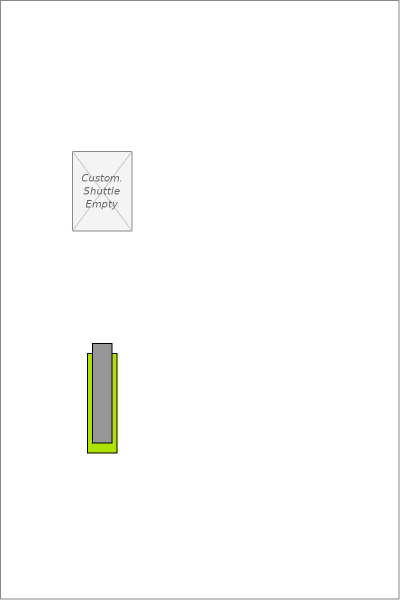
VISUALIZATION VISU_ST170  // 400x600
    Image (72,151 60x80), angle 90, invisible if: NOT __ISVALIDREF(GVL.st170_aut._Mover), image: Custom.Shuttle Empty
    Rectangle (87,353 30x100)
    Rectangle (92,343 20x100)
        p2738717112: -GVL.st170_aut.fb_ABL_RFID.simu_axis170_01Z.rOUT_PixActual
END_VISUALIZATION

// ---- POUs/20_AUTO/ST175/VISU_Recipe_ST175.TcVIS
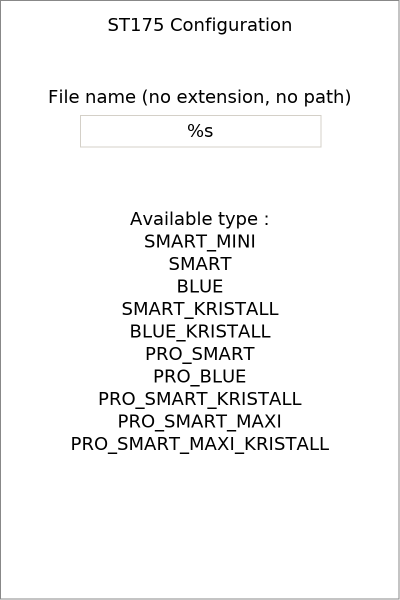
VISUALIZATION VISU_Recipe_ST175  // 400x600
    Textfield (80,115 241x32), "%s", text variable: _20_AUTO.recipe.st175.file_name
        OnMouseDown: write the text variable via Default
    Label (0,5 400x40), "ST175 Configuration"
    Label (24,87 352x20), "File name (no extension, no path)"
    Label (59,177 282x309), "Available type : SMART_MINI SMART BLUE SMART_KRISTALL BLUE_KRISTALL PRO_SMART PRO_BLUE PRO_SMART_KRISTALL PRO_SMART_MAXI PRO_SMART_MAXI_KRISTALL"
END_VISUALIZATION

// ---- POUs/20_AUTO/ST180/VISU_Recipe_ST180.TcVIS
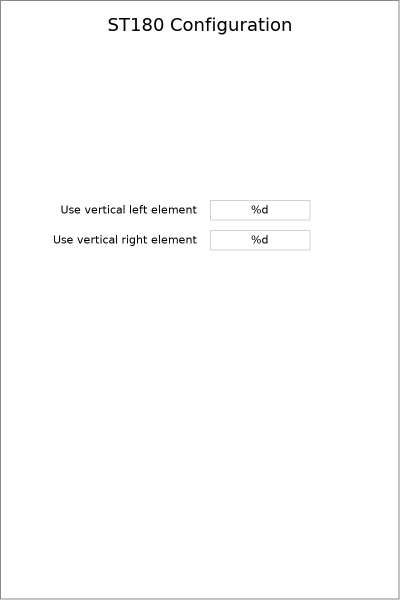
VISUALIZATION VISU_Recipe_ST180  // 400x600
    Label (0,5 400x40), "ST180 Configuration"
    Label (0,200 200x20), "Use vertical left element"
    Label (0,230 200x20), "Use vertical right element"
    Textfield (210,200 100x20), "%d", text variable: _20_AUTO.recipe.st180.xUseVerLeft
        OnMouseDown: write the text variable via Default
    Textfield (210,230 100x20), "%d", text variable: _20_AUTO.recipe.st180.xUseVerRight
        OnMouseDown: write the text variable via Default
END_VISUALIZATION

// ---- POUs/20_AUTO/ST180/VISU_ST180.TcVIS
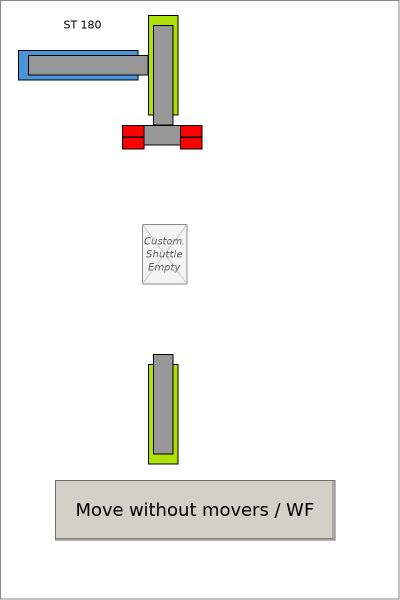
VISUALIZATION VISU_ST180  // 400x600
    Image (142,224 45x60), invisible if: NOT __ISVALIDREF(GVL.st180_aut._Mover), image: Custom.Shuttle Empty
    Rectangle (18,50 120x30)
    Rectangle (28,55 120x20)
        p3560616238: GVL.st180_aut.fb_Pnp.fb_simu_axis180_01Y.rOUT_PixActual
    Rectangle (148,15 30x100)
        p3560616238: GVL.st180_aut.fb_Pnp.fb_simu_axis180_01Y.rOUT_PixActual
    Rectangle (153,25 20x100)
        p2738717112: GVL.st180_aut.fb_Pnp.fb_simu_axis180_02Z.rOUT_PixActual
        p3560616238: GVL.st180_aut.fb_Pnp.fb_simu_axis180_01Y.rOUT_PixActual
    Label (40,15 85x20), "ST 180"
    Rectangle (122,125 80x20)
        p2738717112: GVL.st180_aut.fb_Pnp.fb_simu_axis180_02Z.rOUT_PixActual
        p3560616238: GVL.st180_aut.fb_Pnp.fb_simu_axis180_01Y.rOUT_PixActual
    Ellipse (123,125 20x20), colour toggle: GVL.st180_aut.fb_Pnp.fb_griperLeft.xIN_GS
        p3560616238: GVL.st180_aut.fb_Pnp.fb_simu_axis180_01Y.rOUT_PixActual
        p2738717112: GVL.st180_aut.fb_Pnp.fb_simu_axis180_02Z.rOUT_PixActual
    Ellipse (181,125 20x20), colour toggle: GVL.st180_aut.fb_Pnp.fb_griperRight.xIN_GS
        p3560616238: GVL.st180_aut.fb_Pnp.fb_simu_axis180_01Y.rOUT_PixActual
        p2738717112: GVL.st180_aut.fb_Pnp.fb_simu_axis180_02Z.rOUT_PixActual
    Rectangle (122,125 22x12), invisible if: NOT GVL.st180_aut.fb_Pnp.fb_clampLeft.xIN_GS
        p3560616238: GVL.st180_aut.fb_Pnp.fb_simu_axis180_01Y.rOUT_PixActual
        p2738717112: GVL.st180_aut.fb_Pnp.fb_simu_axis180_02Z.rOUT_PixActual
    Rectangle (180,125 22x12), invisible if: NOT GVL.st180_aut.fb_Pnp.fb_clampRight.xIN_GS
        p3560616238: GVL.st180_aut.fb_Pnp.fb_simu_axis180_01Y.rOUT_PixActual
        p2738717112: GVL.st180_aut.fb_Pnp.fb_simu_axis180_02Z.rOUT_PixActual
    Rectangle (122,137 22x12), invisible if: NOT GVL.st180_aut.fb_Pnp.fb_clampLeft.xIN_AS
        p3560616238: GVL.st180_aut.fb_Pnp.fb_simu_axis180_01Y.rOUT_PixActual
        p2738717112: GVL.st180_aut.fb_Pnp.fb_simu_axis180_02Z.rOUT_PixActual
    Rectangle (180,137 22x12), invisible if: NOT GVL.st180_aut.fb_Pnp.fb_clampRight.xIN_AS
        p3560616238: GVL.st180_aut.fb_Pnp.fb_simu_axis180_01Y.rOUT_PixActual
        p2738717112: GVL.st180_aut.fb_Pnp.fb_simu_axis180_02Z.rOUT_PixActual
    Rectangle (148,364 30x100)
    Rectangle (153,354 20x100)
        p2738717112: -GVL.st180_aut.fb_Pnp.fb_simu_axis180_10Z.rOUT_PixActual
    Button (55,480 280x60), "Move without movers / WF", colour toggle: HMI.bArForceCyclusState[StationList_e.ST180]
        tap HMI.btArForceCyclus[StationList_e.ST180].button
END_VISUALIZATION

// ---- POUs/20_AUTO/ST185/VISU_Recipe_ST185.TcVIS
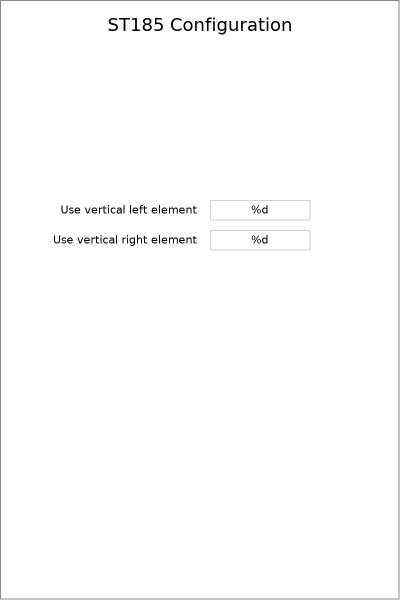
VISUALIZATION VISU_Recipe_ST185  // 400x600
    Label (0,5 400x40), "ST185 Configuration"
    Label (0,200 200x20), "Use vertical left element"
    Label (0,230 200x20), "Use vertical right element"
    Textfield (210,200 100x20), "%d", text variable: _20_AUTO.recipe.st185.xUseVerLeft
        OnMouseDown: write the text variable via Default
    Textfield (210,230 100x20), "%d", text variable: _20_AUTO.recipe.st185.xUseVerRight
        OnMouseDown: write the text variable via Default
END_VISUALIZATION

// ---- VISUs/VISU_LinearConfigArray.TcVIS
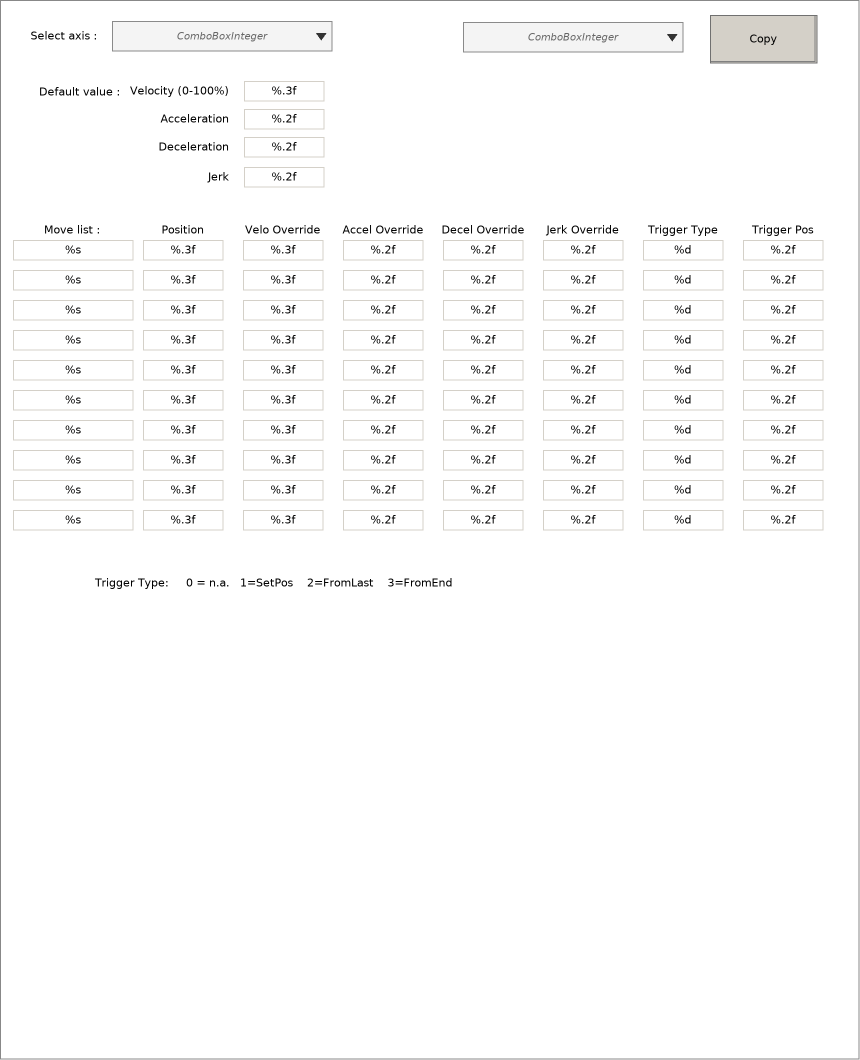
VISUALIZATION VISU_LinearConfigArray  // 860x1060
    Label (25,220 94x20), "Move list :"
    Label (12,82 135x20), "Default value :"
    Label (22,21 84x30), "Select axis :"
    Label (132,81 100x20), "Velocity (0-100%)"
    Label (132,109 100x20), "Acceleration"
    Label (132,137 100x20), "Deceleration"
    Label (132,167 100x20), "Jerk"
    Textfield (244,81 80x20), "%.3f", text variable: _20_AUTO.recipe.linearAxis[HMI.iSelectAxis].defProfile.lrVelocity
        OnMouseDown: write the text variable via Default
    Textfield (244,109 80x20), "%.2f", text variable: _20_AUTO.recipe.linearAxis[HMI.iSelectAxis].defProfile.lrAccel
        OnMouseDown: write the text variable via Default
    Textfield (244,137 80x20), "%.2f", text variable: _20_AUTO.recipe.linearAxis[HMI.iSelectAxis].defProfile.lrDecel
        OnMouseDown: write the text variable via Default
    Textfield (244,167 80x20), "%.2f", text variable: _20_AUTO.recipe.linearAxis[HMI.iSelectAxis].defProfile.lrJerk
        OnMouseDown: write the text variable via Default
    Label (233,220 100x20), "Velo Override"
    Label (333,220 100x20), "Accel Override"
    Label (433,220 100x20), "Decel Override"
    Label (533,220 100x20), "Jerk Override"
    Label (633,220 100x20), "Trigger Type"
    Label (733,220 100x20), "Trigger Pos"
    Textfield (243,240 80x20), "%.3f", text variable: _20_AUTO.recipe.linearAxis[HMI.iSelectAxis].movesList[0].lrVelocity
        OnMouseDown: write the text variable via Default
    Textfield (343,240 80x20), "%.2f", text variable: _20_AUTO.recipe.linearAxis[HMI.iSelectAxis].movesList[0].lrAccel
        OnMouseDown: write the text variable via Default
    Textfield (443,240 80x20), "%.2f", text variable: _20_AUTO.recipe.linearAxis[HMI.iSelectAxis].movesList[0].lrDecel
        OnMouseDown: write the text variable via Default
    Textfield (543,240 80x20), "%.2f", text variable: _20_AUTO.recipe.linearAxis[HMI.iSelectAxis].movesList[0].lrJerk
        OnMouseDown: write the text variable via Default
    Textfield (643,240 80x20), "%d", text variable: _20_AUTO.recipe.linearAxis[HMI.iSelectAxis].movesList[0].TriggerType
        OnMouseDown: write the text variable via Default
    Textfield (743,240 80x20), "%.2f", text variable: _20_AUTO.recipe.linearAxis[HMI.iSelectAxis].movesList[0].TriggerPos
        OnMouseDown: write the text variable via Default
    Textfield (243,270 80x20), "%.3f", text variable: _20_AUTO.recipe.linearAxis[HMI.iSelectAxis].movesList[1].lrVelocity
        OnMouseDown: write the text variable via Default
    Textfield (343,270 80x20), "%.2f", text variable: _20_AUTO.recipe.linearAxis[HMI.iSelectAxis].movesList[1].lrAccel
        OnMouseDown: write the text variable via Default
    Textfield (443,270 80x20), "%.2f", text variable: _20_AUTO.recipe.linearAxis[HMI.iSelectAxis].movesList[1].lrDecel
        OnMouseDown: write the text variable via Default
    Textfield (543,270 80x20), "%.2f", text variable: _20_AUTO.recipe.linearAxis[HMI.iSelectAxis].movesList[1].lrJerk
        OnMouseDown: write the text variable via Default
    Textfield (643,270 80x20), "%d", text variable: _20_AUTO.recipe.linearAxis[HMI.iSelectAxis].movesList[1].TriggerType
        OnMouseDown: write the text variable via Default
    Textfield (743,270 80x20), "%.2f", text variable: _20_AUTO.recipe.linearAxis[HMI.iSelectAxis].movesList[1].TriggerPos
        OnMouseDown: write the text variable via Default
    Textfield (243,300 80x20), "%.3f", text variable: _20_AUTO.recipe.linearAxis[HMI.iSelectAxis].movesList[2].lrVelocity
        OnMouseDown: write the text variable via Default
    Textfield (343,300 80x20), "%.2f", text variable: _20_AUTO.recipe.linearAxis[HMI.iSelectAxis].movesList[2].lrAccel
        OnMouseDown: write the text variable via Default
    Textfield (443,300 80x20), "%.2f", text variable: _20_AUTO.recipe.linearAxis[HMI.iSelectAxis].movesList[2].lrDecel
        OnMouseDown: write the text variable via Default
    Textfield (543,300 80x20), "%.2f", text variable: _20_AUTO.recipe.linearAxis[HMI.iSelectAxis].movesList[2].lrJerk
        OnMouseDown: write the text variable via Default
    Textfield (643,300 80x20), "%d", text variable: _20_AUTO.recipe.linearAxis[HMI.iSelectAxis].movesList[2].TriggerType
        OnMouseDown: write the text variable via Default
    Textfield (743,300 80x20), "%.2f", text variable: _20_AUTO.recipe.linearAxis[HMI.iSelectAxis].movesList[2].TriggerPos
        OnMouseDown: write the text variable via Default
    Textfield (243,330 80x20), "%.3f", text variable: _20_AUTO.recipe.linearAxis[HMI.iSelectAxis].movesList[3].lrVelocity
        OnMouseDown: write the text variable via Default
    Textfield (343,330 80x20), "%.2f", text variable: _20_AUTO.recipe.linearAxis[HMI.iSelectAxis].movesList[3].lrAccel
        OnMouseDown: write the text variable via Default
    Textfield (443,330 80x20), "%.2f", text variable: _20_AUTO.recipe.linearAxis[HMI.iSelectAxis].movesList[3].lrDecel
        OnMouseDown: write the text variable via Default
    Textfield (543,330 80x20), "%.2f", text variable: _20_AUTO.recipe.linearAxis[HMI.iSelectAxis].movesList[3].lrJerk
        OnMouseDown: write the text variable via Default
    Textfield (643,330 80x20), "%d", text variable: _20_AUTO.recipe.linearAxis[HMI.iSelectAxis].movesList[3].TriggerType
        OnMouseDown: write the text variable via Default
    Textfield (743,330 80x20), "%.2f", text variable: _20_AUTO.recipe.linearAxis[HMI.iSelectAxis].movesList[3].TriggerPos
        OnMouseDown: write the text variable via Default
    Textfield (243,360 80x20), "%.3f", text variable: _20_AUTO.recipe.linearAxis[HMI.iSelectAxis].movesList[4].lrVelocity
        OnMouseDown: write the text variable via Default
    Textfield (343,360 80x20), "%.2f", text variable: _20_AUTO.recipe.linearAxis[HMI.iSelectAxis].movesList[4].lrAccel
        OnMouseDown: write the text variable via Default
    Textfield (443,360 80x20), "%.2f", text variable: _20_AUTO.recipe.linearAxis[HMI.iSelectAxis].movesList[4].lrDecel
        OnMouseDown: write the text variable via Default
    Textfield (543,360 80x20), "%.2f", text variable: _20_AUTO.recipe.linearAxis[HMI.iSelectAxis].movesList[4].lrJerk
        OnMouseDown: write the text variable via Default
    Textfield (643,360 80x20), "%d", text variable: _20_AUTO.recipe.linearAxis[HMI.iSelectAxis].movesList[4].TriggerType
        OnMouseDown: write the text variable via Default
    Textfield (743,360 80x20), "%.2f", text variable: _20_AUTO.recipe.linearAxis[HMI.iSelectAxis].movesList[4].TriggerPos
        OnMouseDown: write the text variable via Default
    Textfield (243,390 80x20), "%.3f", text variable: _20_AUTO.recipe.linearAxis[HMI.iSelectAxis].movesList[5].lrVelocity
        OnMouseDown: write the text variable via Default
    Textfield (343,390 80x20), "%.2f", text variable: _20_AUTO.recipe.linearAxis[HMI.iSelectAxis].movesList[5].lrAccel
        OnMouseDown: write the text variable via Default
    Textfield (443,390 80x20), "%.2f", text variable: _20_AUTO.recipe.linearAxis[HMI.iSelectAxis].movesList[5].lrDecel
        OnMouseDown: write the text variable via Default
    Textfield (543,390 80x20), "%.2f", text variable: _20_AUTO.recipe.linearAxis[HMI.iSelectAxis].movesList[5].lrJerk
        OnMouseDown: write the text variable via Default
    Textfield (643,390 80x20), "%d", text variable: _20_AUTO.recipe.linearAxis[HMI.iSelectAxis].movesList[5].TriggerType
        OnMouseDown: write the text variable via Default
    Textfield (743,390 80x20), "%.2f", text variable: _20_AUTO.recipe.linearAxis[HMI.iSelectAxis].movesList[5].TriggerPos
        OnMouseDown: write the text variable via Default
    Textfield (243,420 80x20), "%.3f", text variable: _20_AUTO.recipe.linearAxis[HMI.iSelectAxis].movesList[6].lrVelocity
        OnMouseDown: write the text variable via Default
    Textfield (343,420 80x20), "%.2f", text variable: _20_AUTO.recipe.linearAxis[HMI.iSelectAxis].movesList[6].lrAccel
        OnMouseDown: write the text variable via Default
    Textfield (443,420 80x20), "%.2f", text variable: _20_AUTO.recipe.linearAxis[HMI.iSelectAxis].movesList[6].lrDecel
        OnMouseDown: write the text variable via Default
    Textfield (543,420 80x20), "%.2f", text variable: _20_AUTO.recipe.linearAxis[HMI.iSelectAxis].movesList[6].lrJerk
        OnMouseDown: write the text variable via Default
    Textfield (643,420 80x20), "%d", text variable: _20_AUTO.recipe.linearAxis[HMI.iSelectAxis].movesList[6].TriggerType
        OnMouseDown: write the text variable via Default
    Textfield (743,420 80x20), "%.2f", text variable: _20_AUTO.recipe.linearAxis[HMI.iSelectAxis].movesList[6].TriggerPos
        OnMouseDown: write the text variable via Default
    Textfield (243,450 80x20), "%.3f", text variable: _20_AUTO.recipe.linearAxis[HMI.iSelectAxis].movesList[7].lrVelocity
        OnMouseDown: write the text variable via Default
    Textfield (343,450 80x20), "%.2f", text variable: _20_AUTO.recipe.linearAxis[HMI.iSelectAxis].movesList[7].lrAccel
        OnMouseDown: write the text variable via Default
    Textfield (443,450 80x20), "%.2f", text variable: _20_AUTO.recipe.linearAxis[HMI.iSelectAxis].movesList[7].lrDecel
        OnMouseDown: write the text variable via Default
    Textfield (543,450 80x20), "%.2f", text variable: _20_AUTO.recipe.linearAxis[HMI.iSelectAxis].movesList[7].lrJerk
        OnMouseDown: write the text variable via Default
    Textfield (643,450 80x20), "%d", text variable: _20_AUTO.recipe.linearAxis[HMI.iSelectAxis].movesList[7].TriggerType
        OnMouseDown: write the text variable via Default
    Textfield (743,450 80x20), "%.2f", text variable: _20_AUTO.recipe.linearAxis[HMI.iSelectAxis].movesList[7].TriggerPos
        OnMouseDown: write the text variable via Default
    Textfield (243,480 80x20), "%.3f", text variable: _20_AUTO.recipe.linearAxis[HMI.iSelectAxis].movesList[8].lrVelocity
        OnMouseDown: write the text variable via Default
    Textfield (343,480 80x20), "%.2f", text variable: _20_AUTO.recipe.linearAxis[HMI.iSelectAxis].movesList[8].lrAccel
        OnMouseDown: write the text variable via Default
    Textfield (443,480 80x20), "%.2f", text variable: _20_AUTO.recipe.linearAxis[HMI.iSelectAxis].movesList[8].lrDecel
        OnMouseDown: write the text variable via Default
    Textfield (543,480 80x20), "%.2f", text variable: _20_AUTO.recipe.linearAxis[HMI.iSelectAxis].movesList[8].lrJerk
        OnMouseDown: write the text variable via Default
    Textfield (643,480 80x20), "%d", text variable: _20_AUTO.recipe.linearAxis[HMI.iSelectAxis].movesList[8].TriggerType
        OnMouseDown: write the text variable via Default
    Textfield (743,480 80x20), "%.2f", text variable: _20_AUTO.recipe.linearAxis[HMI.iSelectAxis].movesList[8].TriggerPos
        OnMouseDown: write the text variable via Default
    Textfield (243,510 80x20), "%.3f", text variable: _20_AUTO.recipe.linearAxis[HMI.iSelectAxis].movesList[9].lrVelocity
        OnMouseDown: write the text variable via Default
    Textfield (343,510 80x20), "%.2f", text variable: _20_AUTO.recipe.linearAxis[HMI.iSelectAxis].movesList[9].lrAccel
        OnMouseDown: write the text variable via Default
    Textfield (443,510 80x20), "%.2f", text variable: _20_AUTO.recipe.linearAxis[HMI.iSelectAxis].movesList[9].lrDecel
        OnMouseDown: write the text variable via Default
    Textfield (543,510 80x20), "%.2f", text variable: _20_AUTO.recipe.linearAxis[HMI.iSelectAxis].movesList[9].lrJerk
        OnMouseDown: write the text variable via Default
    Textfield (643,510 80x20), "%d", text variable: _20_AUTO.recipe.linearAxis[HMI.iSelectAxis].movesList[9].TriggerType
        OnMouseDown: write the text variable via Default
    Textfield (743,510 80x20), "%.2f", text variable: _20_AUTO.recipe.linearAxis[HMI.iSelectAxis].movesList[9].TriggerPos
        OnMouseDown: write the text variable via Default
    ComboBoxInteger (112,21 220x30), variable: HMI.iSelectAxis
    Label (133,220 100x20), "Position"
    Textfield (143,240 80x20), "%.3f", text variable: _20_AUTO.recipe.linearAxis[HMI.iSelectAxis].movesList[0].lrPosition
        OnMouseDown: write the text variable via Default
    Textfield (143,270 80x20), "%.3f", text variable: _20_AUTO.recipe.linearAxis[HMI.iSelectAxis].movesList[1].lrPosition
        OnMouseDown: write the text variable via Default
    Textfield (143,300 80x20), "%.3f", text variable: _20_AUTO.recipe.linearAxis[HMI.iSelectAxis].movesList[2].lrPosition
        OnMouseDown: write the text variable via Default
    Textfield (143,330 80x20), "%.3f", text variable: _20_AUTO.recipe.linearAxis[HMI.iSelectAxis].movesList[3].lrPosition
        OnMouseDown: write the text variable via Default
    Textfield (143,360 80x20), "%.3f", text variable: _20_AUTO.recipe.linearAxis[HMI.iSelectAxis].movesList[4].lrPosition
        OnMouseDown: write the text variable via Default
    Textfield (143,390 80x20), "%.3f", text variable: _20_AUTO.recipe.linearAxis[HMI.iSelectAxis].movesList[5].lrPosition
        OnMouseDown: write the text variable via Default
    Textfield (143,420 80x20), "%.3f", text variable: _20_AUTO.recipe.linearAxis[HMI.iSelectAxis].movesList[6].lrPosition
        OnMouseDown: write the text variable via Default
    Textfield (143,450 80x20), "%.3f", text variable: _20_AUTO.recipe.linearAxis[HMI.iSelectAxis].movesList[7].lrPosition
        OnMouseDown: write the text variable via Default
    Textfield (143,480 80x20), "%.3f", text variable: _20_AUTO.recipe.linearAxis[HMI.iSelectAxis].movesList[8].lrPosition
        OnMouseDown: write the text variable via Default
    Textfield (143,510 80x20), "%.3f", text variable: _20_AUTO.recipe.linearAxis[HMI.iSelectAxis].movesList[9].lrPosition
        OnMouseDown: write the text variable via Default
    Textfield (13,240 120x20), "%s", text variable: HMI.movesNames[HMI.iSelectAxis][0]
    Textfield (13,270 120x20), "%s", text variable: HMI.movesNames[HMI.iSelectAxis][1]
    Textfield (13,300 120x20), "%s", text variable: HMI.movesNames[HMI.iSelectAxis][2]
    Textfield (13,330 120x20), "%s", text variable: HMI.movesNames[HMI.iSelectAxis][3]
    Textfield (13,360 120x20), "%s", text variable: HMI.movesNames[HMI.iSelectAxis][4]
    Textfield (13,390 120x20), "%s", text variable: HMI.movesNames[HMI.iSelectAxis][5]
    Textfield (13,420 120x20), "%s", text variable: HMI.movesNames[HMI.iSelectAxis][6]
    Textfield (13,450 120x20), "%s", text variable: HMI.movesNames[HMI.iSelectAxis][7]
    Textfield (13,480 120x20), "%s", text variable: HMI.movesNames[HMI.iSelectAxis][8]
    Textfield (13,510 120x20), "%s", text variable: HMI.movesNames[HMI.iSelectAxis][9]
    ComboBoxInteger (463,22 220x30), variable: HMI.iSelectAxisCopy
    Button (710,15 107x48), "Copy"
        tap HMI.btCopyAxisCfg.button
    Label (56,573 436x20), "Trigger Type: 0 = n.a. 1=SetPos 2=FromLast 3=FromEnd"
END_VISUALIZATION

// ---- VISUs/VISU_Cylinder2PosConfig.TcVIS
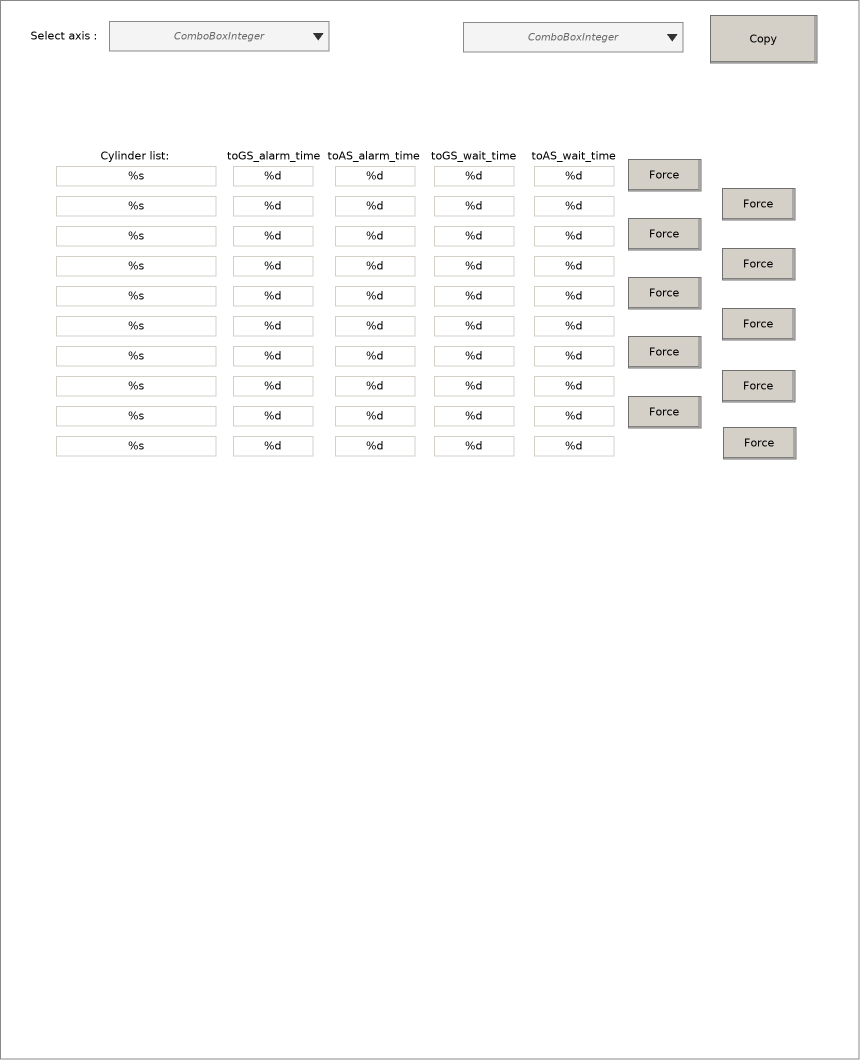
VISUALIZATION VISU_Cylinder2PosConfig  // 860x1060
    Label (88,146 94x20), "Cylinder list:"
    Label (22,21 84x30), "Select axis :"
    Label (324,146 100x20), "toAS_alarm_time"
    Label (424,146 100x20), "toGS_wait_time"
    Label (524,146 100x20), "toAS_wait_time"
    ComboBoxInteger (109,21 220x30), variable: HMI.iSelectCylinder
    Label (224,146 100x20), "toGS_alarm_time"
    Textfield (56,166 160x20), "%s", text variable: HMI.cylinderNames[HMI.iSelectCylinder][0]
    Textfield (56,196 160x20), "%s", text variable: HMI.cylinderNames[HMI.iSelectCylinder][1]
    Textfield (56,226 160x20), "%s", text variable: HMI.cylinderNames[HMI.iSelectCylinder][2]
    Textfield (56,256 160x20), "%s", text variable: HMI.cylinderNames[HMI.iSelectCylinder][3]
    Textfield (56,286 160x20), "%s", text variable: HMI.cylinderNames[HMI.iSelectCylinder][4]
    Textfield (56,316 160x20), "%s", text variable: HMI.cylinderNames[HMI.iSelectCylinder][5]
    Textfield (56,346 160x20), "%s", text variable: HMI.cylinderNames[HMI.iSelectCylinder][6]
    Textfield (56,376 160x20), "%s", text variable: HMI.cylinderNames[HMI.iSelectCylinder][7]
    Textfield (56,406 160x20), "%s", text variable: HMI.cylinderNames[HMI.iSelectCylinder][8]
    Textfield (56,436 160x20), "%s", text variable: HMI.cylinderNames[HMI.iSelectCylinder][9]
    ComboBoxInteger (463,22 220x30), variable: HMI.iSelectCylinderCopy
    Button (710,15 107x48), "Copy"
        tap HMI.btCopyCylinderCfg.button
    Textfield (233,166 80x20), "%d", text variable: _20_AUTO.recipe.cylinder2Pos[HMI.iSelectCylinder][0].toGS_alarm_time
        OnMouseDown: write the text variable via Default
    Textfield (335,166 80x20), "%d", text variable: _20_AUTO.recipe.cylinder2Pos[HMI.iSelectCylinder][0].toAS_alarm_time
        OnMouseDown: write the text variable via Default
    Textfield (434,166 80x20), "%d", text variable: _20_AUTO.recipe.cylinder2Pos[HMI.iSelectCylinder][0].toGS_wait_time
        OnMouseDown: write the text variable via Default
    Textfield (534,166 80x20), "%d", text variable: _20_AUTO.recipe.cylinder2Pos[HMI.iSelectCylinder][0].toAS_wait_time
        OnMouseDown: write the text variable via Default
    Textfield (233,196 80x20), "%d", text variable: _20_AUTO.recipe.cylinder2Pos[HMI.iSelectCylinder][1].toGS_alarm_time
        OnMouseDown: write the text variable via Default
    Textfield (335,196 80x20), "%d", text variable: _20_AUTO.recipe.cylinder2Pos[HMI.iSelectCylinder][1].toAS_alarm_time
        OnMouseDown: write the text variable via Default
    Textfield (434,196 80x20), "%d", text variable: _20_AUTO.recipe.cylinder2Pos[HMI.iSelectCylinder][1].toGS_wait_time
        OnMouseDown: write the text variable via Default
    Textfield (534,196 80x20), "%d", text variable: _20_AUTO.recipe.cylinder2Pos[HMI.iSelectCylinder][1].toAS_wait_time
        OnMouseDown: write the text variable via Default
    Textfield (233,226 80x20), "%d", text variable: _20_AUTO.recipe.cylinder2Pos[HMI.iSelectCylinder][2].toGS_alarm_time
        OnMouseDown: write the text variable via Default
    Textfield (335,226 80x20), "%d", text variable: _20_AUTO.recipe.cylinder2Pos[HMI.iSelectCylinder][2].toAS_alarm_time
        OnMouseDown: write the text variable via Default
    Textfield (434,226 80x20), "%d", text variable: _20_AUTO.recipe.cylinder2Pos[HMI.iSelectCylinder][2].toGS_wait_time
        OnMouseDown: write the text variable via Default
    Textfield (534,226 80x20), "%d", text variable: _20_AUTO.recipe.cylinder2Pos[HMI.iSelectCylinder][2].toAS_wait_time
        OnMouseDown: write the text variable via Default
    Textfield (233,256 80x20), "%d", text variable: _20_AUTO.recipe.cylinder2Pos[HMI.iSelectCylinder][3].toGS_alarm_time
        OnMouseDown: write the text variable via Default
    Textfield (335,256 80x20), "%d", text variable: _20_AUTO.recipe.cylinder2Pos[HMI.iSelectCylinder][3].toAS_alarm_time
        OnMouseDown: write the text variable via Default
    Textfield (434,256 80x20), "%d", text variable: _20_AUTO.recipe.cylinder2Pos[HMI.iSelectCylinder][3].toGS_wait_time
        OnMouseDown: write the text variable via Default
    Textfield (534,256 80x20), "%d", text variable: _20_AUTO.recipe.cylinder2Pos[HMI.iSelectCylinder][3].toAS_wait_time
        OnMouseDown: write the text variable via Default
    Textfield (233,286 80x20), "%d", text variable: _20_AUTO.recipe.cylinder2Pos[HMI.iSelectCylinder][4].toGS_alarm_time
        OnMouseDown: write the text variable via Default
    Textfield (335,286 80x20), "%d", text variable: _20_AUTO.recipe.cylinder2Pos[HMI.iSelectCylinder][4].toAS_alarm_time
        OnMouseDown: write the text variable via Default
    Textfield (434,286 80x20), "%d", text variable: _20_AUTO.recipe.cylinder2Pos[HMI.iSelectCylinder][4].toGS_wait_time
        OnMouseDown: write the text variable via Default
    Textfield (534,286 80x20), "%d", text variable: _20_AUTO.recipe.cylinder2Pos[HMI.iSelectCylinder][4].toAS_wait_time
        OnMouseDown: write the text variable via Default
    Textfield (233,316 80x20), "%d", text variable: _20_AUTO.recipe.cylinder2Pos[HMI.iSelectCylinder][5].toGS_alarm_time
        OnMouseDown: write the text variable via Default
    Textfield (335,316 80x20), "%d", text variable: _20_AUTO.recipe.cylinder2Pos[HMI.iSelectCylinder][5].toAS_alarm_time
        OnMouseDown: write the text variable via Default
    Textfield (434,316 80x20), "%d", text variable: _20_AUTO.recipe.cylinder2Pos[HMI.iSelectCylinder][5].toGS_wait_time
        OnMouseDown: write the text variable via Default
    Textfield (534,316 80x20), "%d", text variable: _20_AUTO.recipe.cylinder2Pos[HMI.iSelectCylinder][5].toAS_wait_time
        OnMouseDown: write the text variable via Default
    Textfield (233,346 80x20), "%d", text variable: _20_AUTO.recipe.cylinder2Pos[HMI.iSelectCylinder][6].toGS_alarm_time
        OnMouseDown: write the text variable via Default
    Textfield (335,346 80x20), "%d", text variable: _20_AUTO.recipe.cylinder2Pos[HMI.iSelectCylinder][6].toAS_alarm_time
        OnMouseDown: write the text variable via Default
    Textfield (434,346 80x20), "%d", text variable: _20_AUTO.recipe.cylinder2Pos[HMI.iSelectCylinder][6].toGS_wait_time
        OnMouseDown: write the text variable via Default
    Textfield (534,346 80x20), "%d", text variable: _20_AUTO.recipe.cylinder2Pos[HMI.iSelectCylinder][6].toAS_wait_time
        OnMouseDown: write the text variable via Default
    Textfield (233,376 80x20), "%d", text variable: _20_AUTO.recipe.cylinder2Pos[HMI.iSelectCylinder][7].toGS_alarm_time
        OnMouseDown: write the text variable via Default
    Textfield (335,376 80x20), "%d", text variable: _20_AUTO.recipe.cylinder2Pos[HMI.iSelectCylinder][7].toAS_alarm_time
        OnMouseDown: write the text variable via Default
    Textfield (434,376 80x20), "%d", text variable: _20_AUTO.recipe.cylinder2Pos[HMI.iSelectCylinder][7].toGS_wait_time
        OnMouseDown: write the text variable via Default
    Textfield (534,376 80x20), "%d", text variable: _20_AUTO.recipe.cylinder2Pos[HMI.iSelectCylinder][7].toAS_wait_time
        OnMouseDown: write the text variable via Default
    Textfield (233,406 80x20), "%d", text variable: _20_AUTO.recipe.cylinder2Pos[HMI.iSelectCylinder][8].toGS_alarm_time
        OnMouseDown: write the text variable via Default
    Textfield (335,406 80x20), "%d", text variable: _20_AUTO.recipe.cylinder2Pos[HMI.iSelectCylinder][8].toAS_alarm_time
        OnMouseDown: write the text variable via Default
    Textfield (434,406 80x20), "%d", text variable: _20_AUTO.recipe.cylinder2Pos[HMI.iSelectCylinder][8].toGS_wait_time
        OnMouseDown: write the text variable via Default
    Textfield (534,406 80x20), "%d", text variable: _20_AUTO.recipe.cylinder2Pos[HMI.iSelectCylinder][8].toAS_wait_time
        OnMouseDown: write the text variable via Default
    Textfield (233,436 80x20), "%d", text variable: _20_AUTO.recipe.cylinder2Pos[HMI.iSelectCylinder][9].toGS_alarm_time
        OnMouseDown: write the text variable via Default
    Textfield (335,436 80x20), "%d", text variable: _20_AUTO.recipe.cylinder2Pos[HMI.iSelectCylinder][9].toAS_alarm_time
        OnMouseDown: write the text variable via Default
    Textfield (434,436 80x20), "%d", text variable: _20_AUTO.recipe.cylinder2Pos[HMI.iSelectCylinder][9].toGS_wait_time
        OnMouseDown: write the text variable via Default
    Textfield (534,436 80x20), "%d", text variable: _20_AUTO.recipe.cylinder2Pos[HMI.iSelectCylinder][9].toAS_wait_time
        OnMouseDown: write the text variable via Default
    Button (723,427 73x32), "Force", colour toggle: HMI.btManuCylinders[HMI.iSelectCylinder][9].on
        tap HMI.btManuCylinders[HMI.iSelectCylinder][10].button
    Button (628,159 73x32), "Force", colour toggle: HMI.btManuCylinders[HMI.iSelectCylinder][1].on
        tap HMI.btManuCylinders[HMI.iSelectCylinder][1].button
    Button (722,188 73x32), "Force", colour toggle: HMI.btManuCylinders[HMI.iSelectCylinder][2].on
        tap HMI.btManuCylinders[HMI.iSelectCylinder][2].button
    Button (628,218 73x32), "Force", colour toggle: HMI.btManuCylinders[HMI.iSelectCylinder][3].on
        tap HMI.btManuCylinders[HMI.iSelectCylinder][3].button
    Button (722,248 73x32), "Force", colour toggle: HMI.btManuCylinders[HMI.iSelectCylinder][4].on
        tap HMI.btManuCylinders[HMI.iSelectCylinder][4].button
    Button (628,277 73x32), "Force", colour toggle: HMI.btManuCylinders[HMI.iSelectCylinder][5].on
        tap HMI.btManuCylinders[HMI.iSelectCylinder][5].button
    Button (722,308 73x32), "Force", colour toggle: HMI.btManuCylinders[HMI.iSelectCylinder][6].on
        tap HMI.btManuCylinders[HMI.iSelectCylinder][6].button
    Button (628,336 73x32), "Force", colour toggle: HMI.btManuCylinders[HMI.iSelectCylinder][7].on
        tap HMI.btManuCylinders[HMI.iSelectCylinder][7].button
    Button (722,370 73x32), "Force", colour toggle: HMI.btManuCylinders[HMI.iSelectCylinder][8].on
        tap HMI.btManuCylinders[HMI.iSelectCylinder][8].button
    Button (628,396 73x32), "Force", colour toggle: HMI.btManuCylinders[HMI.iSelectCylinder][9].on
        tap HMI.btManuCylinders[HMI.iSelectCylinder][9].button
END_VISUALIZATION

// ---- VISUs/VISU_AxisManual.TcVIS
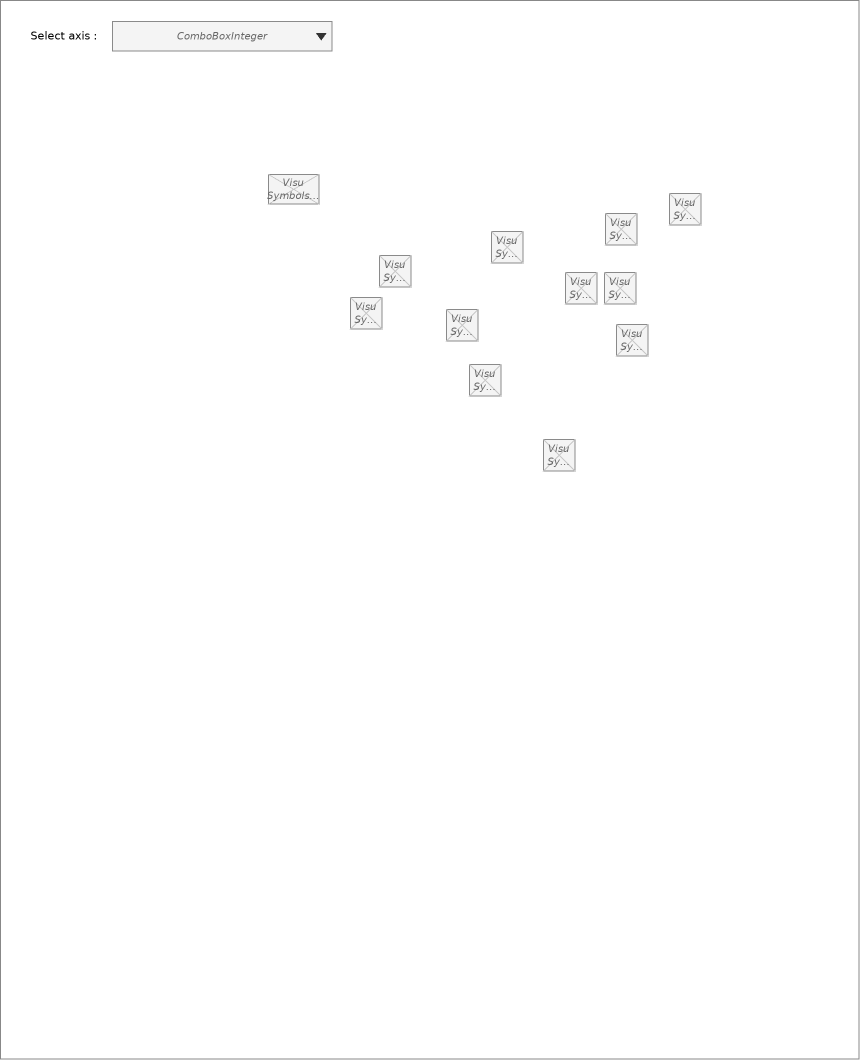
VISUALIZATION VISU_AxisManual  // 860x1060
    Label (22,21 84x30), "Select axis :"
    ComboBoxInteger (112,21 220x30), variable: HMI.iSelectJogAxis
    Image (268,174 51x30), image: VisuSymbols.Symbols.ForwardStandard
    Image (350,297 32x32), image: VisuSymbols.Symbols.Home
    Image (469,364 32x32), image: VisuSymbols.Symbols.Humidity
    Image (543,439 32x32), image: VisuSymbols.Symbols.Keeper
    Image (446,309 32x32), image: VisuSymbols.Symbols.ListNumbers
    Image (604,272 32x32), image: VisuSymbols.Symbols.Marker+
    Image (565,272 32x32), image: VisuSymbols.Symbols.Marker-
    Image (616,324 32x32), image: VisuSymbols.Symbols.Micro
    Image (605,213 32x32), image: VisuSymbols.Symbols.MonitorCurve
    Image (491,231 32x32), image: VisuSymbols.Symbols.Play
    Image (669,193 32x32), image: VisuSymbols.Symbols.Security
    Image (379,255 32x32), image: VisuSymbols.Symbols.Stop
END_VISUALIZATION

// ---- VISUs/VISU_main.TcVIS
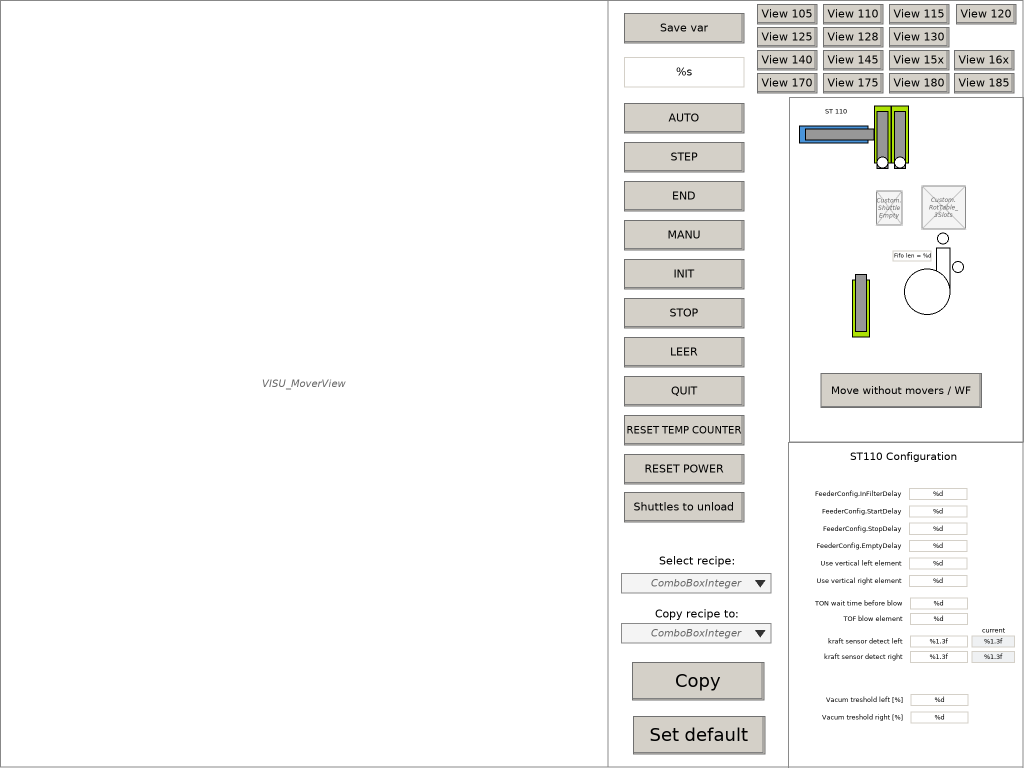
VISUALIZATION VISU_main  // 1024x768
    TabControl (0,0 608x767)
        shows VISU_MoverView()
        shows VISU_LinearConfigArray()
        shows VISU_MoverDetail()
        shows VISU_Cylinder2PosConfig()
        shows VISU_Time()
        [0]: TabTitle=Mover Track, ImageId=Custom.Shuttle Full
        [1]: TabTitle=Linear Axis, ImageId=Custom.RotTable_3Slots
        [2]: TabTitle=Mover details
        [3]: TabTitle=Cylinder config
        [4]: TabTitle=Timing
    Button (624,103 120x30), "AUTO", colour toggle: HMI.btArMain[0].on, input disabled if: HMI.btArMain[0].disable
        tap HMI.btArMain[0].button
    Button (624,142 120x30), "STEP", colour toggle: HMI.btArMain[1].on, input disabled if: HMI.btArMain[1].disable
        tap HMI.btArMain[1].button
    Button (624,181 120x30), "END", colour toggle: HMI.btArMain[2].on, input disabled if: HMI.btArMain[2].disable
        tap HMI.btArMain[2].button
    Button (624,259 120x30), "INIT", colour toggle: HMI.btArMain[4].on, input disabled if: HMI.btArMain[4].disable
        tap HMI.btArMain[4].button
    Button (624,298 120x30), "STOP", colour toggle: HMI.btArMain[5].disable, input disabled if: HMI.btArMain[5].disable
        tap HMI.btArMain[5].button
    Button (624,337 120x30), "LEER", colour toggle: HMI.btArMain[6].disable, input disabled if: HMI.btArMain[6].disable
        tap HMI.btArMain[6].button
    Button (624,376 120x30), "QUIT", colour toggle: HMI.btArMain[7].disable, input disabled if: HMI.btArMain[7].disable
        tap HMI.btArMain[7].button
    Button (624,415 120x30), "RESET TEMP COUNTER", colour toggle: HMI.btArMain[8].disable, input disabled if: HMI.btArMain[8].disable
        tap HMI.btArMain[8].button
    Button (624,220 120x30), "MANU", colour toggle: HMI.btArMain[3].on, input disabled if: HMI.btArMain[3].disable
        tap HMI.btArMain[3].button
    Textfield (624,57 120x30), "%s", text variable: _14_STATE.sStateDbg
    Button (624,454 120x30), "RESET POWER"
        tap HMI.Tast_BL
    Button (624,13 120x30), "Save var", input disabled if: TRUE
        tap FileMan.bSaveData
    Frame (789,97 235x345)
        shows VISU_ST110()
        shows VISU_ST115()
        shows VISU_ST120()
        shows VISU_ST125()
        shows VISU_ST145()
        shows VISU_ST180()
        shows VISU_ST185()
        shows VISU_ST130()
        shows VISU_ST105()
        shows VISU_ST140()
        shows VISU_ST150()
        shows VISU_ST128()
        shows VISU_ST160()
        shows VISU_ST170()
        shows VISU_ST175()
    Button (889,4 60x20), "View 115"
        OnMouseDown: FrameSelectionChange Selection=SelectedFrame=06e07b94-3d2f-4429-a7a0-840881734514, Selection=1, GlobSel=AssignType=Directly, SelType=Locally
        OnMouseDown: FrameSelectionChange Selection=SelectedFrame=9156b980-1735-4d37-9321-1bea537ecf5c, Selection=1, GlobSel=AssignType=Directly, SelType=Locally
    Button (823,4 60x20), "View 110"
        OnMouseDown: FrameSelectionChange Selection=SelectedFrame=06e07b94-3d2f-4429-a7a0-840881734514, GlobSel=AssignType=Directly, SelType=Locally
        OnMouseDown: FrameSelectionChange Selection=SelectedFrame=9156b980-1735-4d37-9321-1bea537ecf5c, GlobSel=AssignType=Directly, SelType=Locally
    Button (956,4 60x20), "View 120"
        OnMouseDown: FrameSelectionChange Selection=SelectedFrame=06e07b94-3d2f-4429-a7a0-840881734514, Selection=2, GlobSel=AssignType=Directly, SelType=Locally
        OnMouseDown: FrameSelectionChange Selection=SelectedFrame=9156b980-1735-4d37-9321-1bea537ecf5c, Selection=2, GlobSel=AssignType=Directly, SelType=Locally
    Frame (788,442 235x347)
        shows VISU_Recipe_ST110()
        shows VISU_Recipe_ST115()
        shows VISU_Recipe_ST120()
        shows VISU_Recipe_ST125()
        shows VISU_Recipe_ST145()
        shows VISU_Recipe_ST180()
        shows VISU_Recipe_ST185()
        shows VISU_Recipe_ST130()
        shows VISU_Recipe_ST105()
        shows VISU_Recipe_ST140()
        shows VISU_Recipe_ST150()
        shows VISU_Recipe_ST128()
        shows VISU_Recipe_ST160()
        shows VISU_Recipe_ST170()
        shows VISU_Recipe_ST175()
    Button (757,27 60x20), "View 125"
        OnMouseDown: FrameSelectionChange Selection=SelectedFrame=06e07b94-3d2f-4429-a7a0-840881734514, Selection=3, GlobSel=AssignType=Directly, SelType=Locally
        OnMouseDown: FrameSelectionChange Selection=SelectedFrame=9156b980-1735-4d37-9321-1bea537ecf5c, Selection=3, GlobSel=AssignType=Directly, SelType=Locally
    ComboBoxInteger (621,573 150x20), variable: PERS.eRecipeCurrent
    Label (622,604 150x20), "Copy recipe to:"
    ComboBoxInteger (621,623 150x20), variable: _20_AUTO.iRecipeCopyDest
    Button (633,716 132x38), "Set default"
        tap HMI.btSetDefault.button
    Button (823,50 60x20), "View 145"
        OnMouseDown: FrameSelectionChange Selection=SelectedFrame=06e07b94-3d2f-4429-a7a0-840881734514, Selection=4, GlobSel=AssignType=Directly, SelType=Locally
        OnMouseDown: FrameSelectionChange Selection=SelectedFrame=9156b980-1735-4d37-9321-1bea537ecf5c, Selection=4, GlobSel=AssignType=Directly, SelType=Locally
    Label (622,551 150x20), "Select recipe:"
    Button (889,73 60x20), "View 180"
        OnMouseDown: FrameSelectionChange Selection=SelectedFrame=06e07b94-3d2f-4429-a7a0-840881734514, Selection=5, GlobSel=AssignType=Directly, SelType=Locally
        OnMouseDown: FrameSelectionChange Selection=SelectedFrame=9156b980-1735-4d37-9321-1bea537ecf5c, Selection=5, GlobSel=AssignType=Directly, SelType=Locally
    Button (954,73 60x20), "View 185"
        OnMouseDown: FrameSelectionChange Selection=SelectedFrame=06e07b94-3d2f-4429-a7a0-840881734514, Selection=6, GlobSel=AssignType=Directly, SelType=Locally
        OnMouseDown: FrameSelectionChange Selection=SelectedFrame=9156b980-1735-4d37-9321-1bea537ecf5c, Selection=6, GlobSel=AssignType=Directly, SelType=Locally
    Button (889,27 60x20), "View 130"
        OnMouseDown: FrameSelectionChange Selection=SelectedFrame=06e07b94-3d2f-4429-a7a0-840881734514, Selection=7, GlobSel=AssignType=Directly, SelType=Locally
        OnMouseDown: FrameSelectionChange Selection=SelectedFrame=9156b980-1735-4d37-9321-1bea537ecf5c, Selection=7, GlobSel=AssignType=Directly, SelType=Locally
    Button (757,4 60x20), "View 105"
        OnMouseDown: FrameSelectionChange Selection=SelectedFrame=06e07b94-3d2f-4429-a7a0-840881734514, Selection=8, GlobSel=AssignType=Directly, SelType=Locally
        OnMouseDown: FrameSelectionChange Selection=SelectedFrame=9156b980-1735-4d37-9321-1bea537ecf5c, Selection=8, GlobSel=AssignType=Directly, SelType=Locally
    Button (757,50 60x20), "View 140"
        OnMouseDown: FrameSelectionChange Selection=SelectedFrame=06e07b94-3d2f-4429-a7a0-840881734514, Selection=9, GlobSel=AssignType=Directly, SelType=Locally
        OnMouseDown: FrameSelectionChange Selection=SelectedFrame=9156b980-1735-4d37-9321-1bea537ecf5c, Selection=9, GlobSel=AssignType=Directly, SelType=Locally
    Button (889,50 60x20), "View 15x"
        OnMouseDown: FrameSelectionChange Selection=SelectedFrame=06e07b94-3d2f-4429-a7a0-840881734514, Selection=10, GlobSel=AssignType=Directly, SelType=Locally
        OnMouseDown: FrameSelectionChange Selection=SelectedFrame=9156b980-1735-4d37-9321-1bea537ecf5c, Selection=10, GlobSel=AssignType=Directly, SelType=Locally
    Button (823,27 60x20), "View 128"
        OnMouseDown: FrameSelectionChange Selection=SelectedFrame=06e07b94-3d2f-4429-a7a0-840881734514, Selection=11, GlobSel=AssignType=Directly, SelType=Locally
        OnMouseDown: FrameSelectionChange Selection=SelectedFrame=9156b980-1735-4d37-9321-1bea537ecf5c, Selection=11, GlobSel=AssignType=Directly, SelType=Locally
    Button (954,50 60x20), "View 16x"
        OnMouseDown: FrameSelectionChange Selection=SelectedFrame=06e07b94-3d2f-4429-a7a0-840881734514, Selection=12, GlobSel=AssignType=Directly, SelType=Locally
        OnMouseDown: FrameSelectionChange Selection=SelectedFrame=9156b980-1735-4d37-9321-1bea537ecf5c, Selection=12, GlobSel=AssignType=Directly, SelType=Locally
    Button (632,662 132x38), "Copy"
        tap HMI.btCopyRecipe.button
    Button (757,73 60x20), "View 170"
        OnMouseDown: FrameSelectionChange Selection=SelectedFrame=06e07b94-3d2f-4429-a7a0-840881734514, Selection=13, GlobSel=AssignType=Directly, SelType=Locally
        OnMouseDown: FrameSelectionChange Selection=SelectedFrame=9156b980-1735-4d37-9321-1bea537ecf5c, Selection=13, GlobSel=AssignType=Directly, SelType=Locally
    Button (823,73 60x20), "View 175"
        OnMouseDown: FrameSelectionChange Selection=SelectedFrame=06e07b94-3d2f-4429-a7a0-840881734514, Selection=14, GlobSel=AssignType=Directly, SelType=Locally
        OnMouseDown: FrameSelectionChange Selection=SelectedFrame=9156b980-1735-4d37-9321-1bea537ecf5c, Selection=14, GlobSel=AssignType=Directly, SelType=Locally
    Button (624,492 120x30), "Shuttles to unload"
        tap MAIN.MoverMan.HMI_send_all_shuttle_to_unload
END_VISUALIZATION

// ---- VISUs/VISU_Time.TcVIS
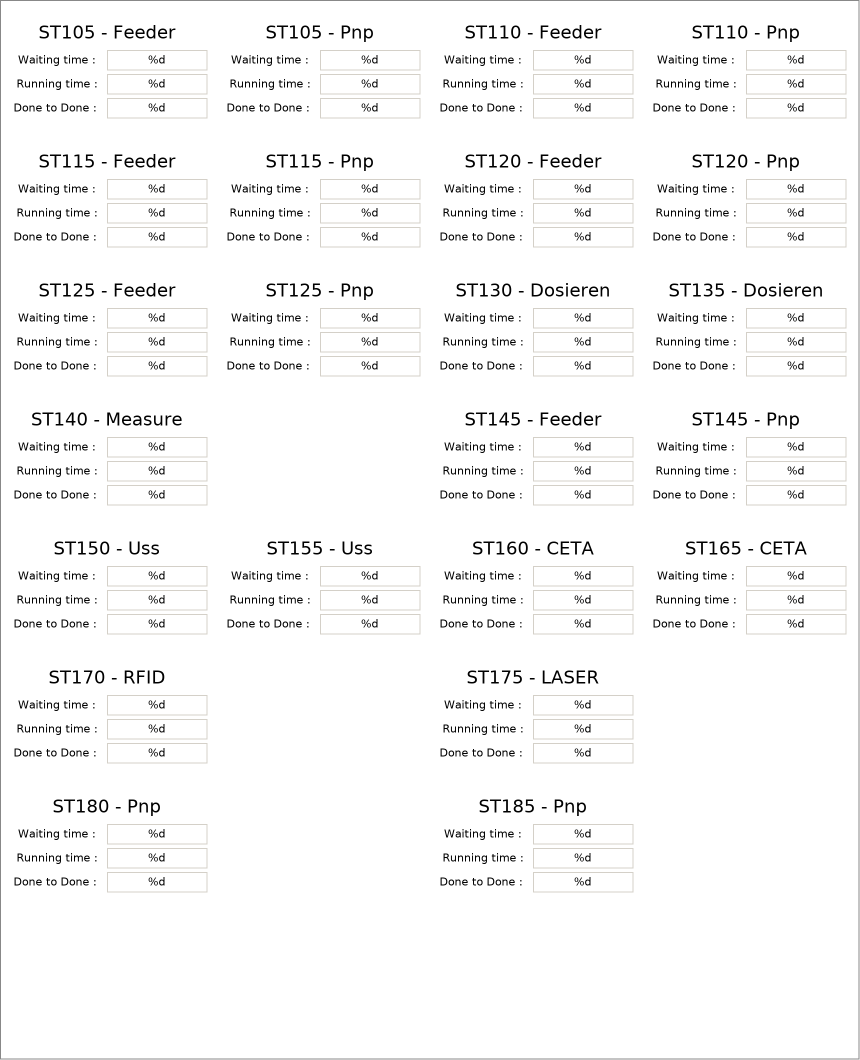
VISUALIZATION VISU_Time  // 860x1060
    Textfield (107,50 100x20), "%d", text variable: GVL.st105_aut.fb_stat_Feeder.tOUT_avgInWait_ms
    Label (7,50 100x20), "Waiting time :"
    Textfield (107,74 100x20), "%d", text variable: GVL.st105_aut.fb_stat_Feeder.tOUT_avgInRun_ms
    Label (7,74 100x20), "Running time :"
    Textfield (107,98 100x20), "%d", text variable: GVL.st105_aut.fb_stat_Feeder.tOUT_avgDoneToDone_ms
    Label (7,98 100x20), "Done to Done :"
    Label (7,19 200x27), "ST105 - Feeder"
    Textfield (320,50 100x20), "%d", text variable: GVL.st105_aut.fb_stat_pnp.tOUT_avgInWait_ms
    Label (220,50 100x20), "Waiting time :"
    Textfield (320,74 100x20), "%d", text variable: GVL.st105_aut.fb_stat_pnp.tOUT_avgInRun_ms
    Label (220,74 100x20), "Running time :"
    Textfield (320,98 100x20), "%d", text variable: GVL.st105_aut.fb_stat_pnp.tOUT_avgDoneToDone_ms
    Label (220,98 100x20), "Done to Done :"
    Label (220,19 200x27), "ST105 - Pnp"
    Textfield (533,50 100x20), "%d", text variable: GVL.st110_aut.fb_stat_Feeder.tOUT_avgInWait_ms
    Label (433,50 100x20), "Waiting time :"
    Textfield (533,74 100x20), "%d", text variable: GVL.st110_aut.fb_stat_Feeder.tOUT_avgInRun_ms
    Label (433,74 100x20), "Running time :"
    Textfield (533,98 100x20), "%d", text variable: GVL.st110_aut.fb_stat_Feeder.tOUT_avgDoneToDone_ms
    Label (433,98 100x20), "Done to Done :"
    Label (433,19 200x27), "ST110 - Feeder"
    Textfield (746,50 100x20), "%d", text variable: GVL.st110_aut.fb_stat_pnp.tOUT_avgInWait_ms
    Label (646,50 100x20), "Waiting time :"
    Textfield (746,74 100x20), "%d", text variable: GVL.st110_aut.fb_stat_pnp.tOUT_avgInRun_ms
    Label (646,74 100x20), "Running time :"
    Textfield (746,98 100x20), "%d", text variable: GVL.st110_aut.fb_stat_pnp.tOUT_avgDoneToDone_ms
    Label (646,98 100x20), "Done to Done :"
    Label (646,19 200x27), "ST110 - Pnp"
    Textfield (107,179 100x20), "%d", text variable: GVL.st115_aut.fb_stat_Feeder.tOUT_avgInWait_ms
    Label (7,179 100x20), "Waiting time :"
    Textfield (107,203 100x20), "%d", text variable: GVL.st115_aut.fb_stat_Feeder.tOUT_avgInRun_ms
    Label (7,203 100x20), "Running time :"
    Textfield (107,227 100x20), "%d", text variable: GVL.st115_aut.fb_stat_Feeder.tOUT_avgDoneToDone_ms
    Label (7,227 100x20), "Done to Done :"
    Label (7,148 200x27), "ST115 - Feeder"
    Textfield (320,179 100x20), "%d", text variable: GVL.st115_aut.fb_stat_pnp.tOUT_avgInWait_ms
    Label (220,179 100x20), "Waiting time :"
    Textfield (320,203 100x20), "%d", text variable: GVL.st115_aut.fb_stat_pnp.tOUT_avgInRun_ms
    Label (220,203 100x20), "Running time :"
    Textfield (320,227 100x20), "%d", text variable: GVL.st115_aut.fb_stat_pnp.tOUT_avgDoneToDone_ms
    Label (220,227 100x20), "Done to Done :"
    Label (220,148 200x27), "ST115 - Pnp"
    Textfield (533,179 100x20), "%d", text variable: GVL.st120_aut.fb_stat_Feeder.tOUT_avgInWait_ms
    Label (433,179 100x20), "Waiting time :"
    Textfield (533,203 100x20), "%d", text variable: GVL.st120_aut.fb_stat_Feeder.tOUT_avgInRun_ms
    Label (433,203 100x20), "Running time :"
    Textfield (533,227 100x20), "%d", text variable: GVL.st120_aut.fb_stat_Feeder.tOUT_avgDoneToDone_ms
    Label (433,227 100x20), "Done to Done :"
    Label (433,148 200x27), "ST120 - Feeder"
    Textfield (746,179 100x20), "%d", text variable: GVL.st120_aut.fb_stat_pnp.tOUT_avgInWait_ms
    Label (646,179 100x20), "Waiting time :"
    Textfield (746,203 100x20), "%d", text variable: GVL.st120_aut.fb_stat_pnp.tOUT_avgInRun_ms
    Label (646,203 100x20), "Running time :"
    Textfield (746,227 100x20), "%d", text variable: GVL.st120_aut.fb_stat_pnp.tOUT_avgDoneToDone_ms
    Label (646,227 100x20), "Done to Done :"
    Label (646,148 200x27), "ST120 - Pnp"
    Textfield (107,308 100x20), "%d", text variable: GVL.st125_aut.fb_stat_Feeder.tOUT_avgInWait_ms
    Label (7,308 100x20), "Waiting time :"
    Textfield (107,332 100x20), "%d", text variable: GVL.st125_aut.fb_stat_Feeder.tOUT_avgInRun_ms
    Label (7,332 100x20), "Running time :"
    Textfield (107,356 100x20), "%d", text variable: GVL.st125_aut.fb_stat_Feeder.tOUT_avgDoneToDone_ms
    Label (7,356 100x20), "Done to Done :"
    Label (7,277 200x27), "ST125 - Feeder"
    Textfield (320,308 100x20), "%d", text variable: GVL.st125_aut.fb_stat_pnp.tOUT_avgInWait_ms
    Label (220,308 100x20), "Waiting time :"
    Textfield (320,332 100x20), "%d", text variable: GVL.st125_aut.fb_stat_pnp.tOUT_avgInRun_ms
    Label (220,332 100x20), "Running time :"
    Textfield (320,356 100x20), "%d", text variable: GVL.st125_aut.fb_stat_pnp.tOUT_avgDoneToDone_ms
    Label (220,356 100x20), "Done to Done :"
    Label (220,277 200x27), "ST125 - Pnp"
    Textfield (533,308 100x20), "%d", text variable: GVL.st130_aut.fb_stat.tOUT_avgInWait_ms
    Label (433,308 100x20), "Waiting time :"
    Textfield (533,332 100x20), "%d", text variable: GVL.st130_aut.fb_stat.tOUT_avgInRun_ms
    Label (433,332 100x20), "Running time :"
    Textfield (533,356 100x20), "%d", text variable: GVL.st130_aut.fb_stat.tOUT_avgDoneToDone_ms
    Label (433,356 100x20), "Done to Done :"
    Label (433,277 200x27), "ST130 - Dosieren"
    Textfield (746,308 100x20), "%d", text variable: GVL.st135_aut.fb_stat.tOUT_avgInWait_ms
    Label (646,308 100x20), "Waiting time :"
    Textfield (746,332 100x20), "%d", text variable: GVL.st135_aut.fb_stat.tOUT_avgInRun_ms
    Label (646,332 100x20), "Running time :"
    Textfield (746,356 100x20), "%d", text variable: GVL.st135_aut.fb_stat.tOUT_avgDoneToDone_ms
    Label (646,356 100x20), "Done to Done :"
    Label (646,277 200x27), "ST135 - Dosieren"
    Textfield (107,437 100x20), "%d", text variable: GVL.st140_aut.fb_stat.tOUT_avgInWait_ms
    Label (7,437 100x20), "Waiting time :"
    Textfield (107,461 100x20), "%d", text variable: GVL.st140_aut.fb_stat.tOUT_avgInRun_ms
    Label (7,461 100x20), "Running time :"
    Textfield (107,485 100x20), "%d", text variable: GVL.st140_aut.fb_stat.tOUT_avgDoneToDone_ms
    Label (7,485 100x20), "Done to Done :"
    Label (7,406 200x27), "ST140 - Measure"
    Textfield (533,437 100x20), "%d", text variable: GVL.st145_aut.fb_stat_Feeder.tOUT_avgInWait_ms
    Label (433,437 100x20), "Waiting time :"
    Textfield (533,461 100x20), "%d", text variable: GVL.st145_aut.fb_stat_Feeder.tOUT_avgInRun_ms
    Label (433,461 100x20), "Running time :"
    Textfield (533,485 100x20), "%d", text variable: GVL.st145_aut.fb_stat_Feeder.tOUT_avgDoneToDone_ms
    Label (433,485 100x20), "Done to Done :"
    Label (433,406 200x27), "ST145 - Feeder"
    Textfield (746,437 100x20), "%d", text variable: GVL.st145_aut.fb_stat_pnp.tOUT_avgInWait_ms
    Label (646,437 100x20), "Waiting time :"
    Textfield (746,461 100x20), "%d", text variable: GVL.st145_aut.fb_stat_pnp.tOUT_avgInRun_ms
    Label (646,461 100x20), "Running time :"
    Textfield (746,485 100x20), "%d", text variable: GVL.st145_aut.fb_stat_pnp.tOUT_avgDoneToDone_ms
    Label (646,485 100x20), "Done to Done :"
    Label (646,406 200x27), "ST145 - Pnp"
    Textfield (107,566 100x20), "%d", text variable: GVL.st150_aut.fb_stat.tOUT_avgInWait_ms
    Label (7,566 100x20), "Waiting time :"
    Textfield (107,590 100x20), "%d", text variable: GVL.st150_aut.fb_stat.tOUT_avgInRun_ms
    Label (7,590 100x20), "Running time :"
    Textfield (107,614 100x20), "%d", text variable: GVL.st150_aut.fb_stat.tOUT_avgDoneToDone_ms
    Label (7,614 100x20), "Done to Done :"
    Label (7,535 200x27), "ST150 - Uss"
    Textfield (320,566 100x20), "%d", text variable: GVL.st155_aut.fb_stat.tOUT_avgInWait_ms
    Label (220,566 100x20), "Waiting time :"
    Textfield (320,590 100x20), "%d", text variable: GVL.st155_aut.fb_stat.tOUT_avgInRun_ms
    Label (220,590 100x20), "Running time :"
    Textfield (320,614 100x20), "%d", text variable: GVL.st155_aut.fb_stat.tOUT_avgDoneToDone_ms
    Label (220,614 100x20), "Done to Done :"
    Label (220,535 200x27), "ST155 - Uss"
    Textfield (533,566 100x20), "%d", text variable: GVL.st160_aut.fb_stat.tOUT_avgInWait_ms
    Label (433,566 100x20), "Waiting time :"
    Textfield (533,590 100x20), "%d", text variable: GVL.st160_aut.fb_stat.tOUT_avgInRun_ms
    Label (433,590 100x20), "Running time :"
    Textfield (533,614 100x20), "%d", text variable: GVL.st160_aut.fb_stat.tOUT_avgDoneToDone_ms
    Label (433,614 100x20), "Done to Done :"
    Label (433,535 200x27), "ST160 - CETA"
    Textfield (746,566 100x20), "%d", text variable: GVL.st165_aut.fb_stat.tOUT_avgInWait_ms
    Label (646,566 100x20), "Waiting time :"
    Textfield (746,590 100x20), "%d", text variable: GVL.st165_aut.fb_stat.tOUT_avgInRun_ms
    Label (646,590 100x20), "Running time :"
    Textfield (746,614 100x20), "%d", text variable: GVL.st165_aut.fb_stat.tOUT_avgDoneToDone_ms
    Label (646,614 100x20), "Done to Done :"
    Label (646,535 200x27), "ST165 - CETA"
    Textfield (107,695 100x20), "%d", text variable: GVL.st170_aut.fb_stat.tOUT_avgInWait_ms
    Label (7,695 100x20), "Waiting time :"
    Textfield (107,719 100x20), "%d", text variable: GVL.st170_aut.fb_stat.tOUT_avgInRun_ms
    Label (7,719 100x20), "Running time :"
    Textfield (107,743 100x20), "%d", text variable: GVL.st170_aut.fb_stat.tOUT_avgDoneToDone_ms
    Label (7,743 100x20), "Done to Done :"
    Label (7,664 200x27), "ST170 - RFID"
    Textfield (533,695 100x20), "%d", text variable: GVL.st175_aut.fb_stat.tOUT_avgInWait_ms
    Label (433,695 100x20), "Waiting time :"
    Textfield (533,719 100x20), "%d", text variable: GVL.st175_aut.fb_stat.tOUT_avgInRun_ms
    Label (433,719 100x20), "Running time :"
    Textfield (533,743 100x20), "%d", text variable: GVL.st175_aut.fb_stat.tOUT_avgDoneToDone_ms
    Label (433,743 100x20), "Done to Done :"
    Label (433,664 200x27), "ST175 - LASER"
    Textfield (107,824 100x20), "%d", text variable: GVL.st180_aut.fb_stat.tOUT_avgInWait_ms
    Label (7,824 100x20), "Waiting time :"
    Textfield (107,848 100x20), "%d", text variable: GVL.st180_aut.fb_stat.tOUT_avgInRun_ms
    Label (7,848 100x20), "Running time :"
    Textfield (107,872 100x20), "%d", text variable: GVL.st180_aut.fb_stat.tOUT_avgDoneToDone_ms
    Label (7,872 100x20), "Done to Done :"
    Label (7,793 200x27), "ST180 - Pnp"
    Textfield (533,824 100x20), "%d", text variable: GVL.st185_aut.fb_stat.tOUT_avgInWait_ms
    Label (433,824 100x20), "Waiting time :"
    Textfield (533,848 100x20), "%d", text variable: GVL.st185_aut.fb_stat.tOUT_avgInRun_ms
    Label (433,848 100x20), "Running time :"
    Textfield (533,872 100x20), "%d", text variable: GVL.st185_aut.fb_stat.tOUT_avgDoneToDone_ms
    Label (433,872 100x20), "Done to Done :"
    Label (433,793 200x27), "ST185 - Pnp"
END_VISUALIZATION
